VAR_GLOBAL
	stTempLoad				: ST_TempLoad;
	stTempSave				: ST_TempSave;
END_VAR

(* stored: Version 1.1.0.1, ProductVersion 3.1.4024.12
   GVL GVL_20_Application: Id {44b4d13a-449a-4cf8-9d7f-415bf0aea4b6} *)
